// TIA Portal project "lab6" (V15)

(* hardware
DEVICE "S7-1200 station_1"  S7-1200 Station
   slot 0: "Rack_0"  S7-1200 Rack  Rack  V1.0
   slot 1: "PLC_1"  CPU 1214C DC/DC/DC  6ES7 214-1AG40-0XB0  V4.2
      slot 3: "AQ 1x12BIT_1"  AQ1 signal board  6ES7 232-4HA30-0XB0  V1.0
   slot 101: "CM 1243-5"  CM 1243-5  6GK7 243-5DX30-0XE0  V1.3
   slot 102: "CM 1241 (RS485)_1"  CM 1241 (RS485)  6ES7 241-1CH30-0XB0  V1.0
*)

// ===== PLC "PLC_1"  CPU 1214C DC/DC/DC =====

VAR_GLOBAL   // PLC tag table "Default tag table"
   "Tag_1" AT %I0.0 : Bool;
   "Tag_2" AT %MW10 : Int;
   "Tag_3" AT %Q0.5 : Bool;
   "Tag_4" AT %I0.1 : Bool;
   "Tag_5" AT %Q0.1 : Bool;
   "Tag_6" AT %Q0.2 : Bool;
   "System_Byte" AT %MB1 : Byte;
   "FirstScan" AT %M1.0 : Bool;
   "DiagStatusUpdate" AT %M1.1 : Bool;
   "AlwaysTRUE" AT %M1.2 : Bool;
   "AlwaysFALSE" AT %M1.3 : Bool;
   "Clock_Byte" AT %MB0 : Byte;
   "Clock_10Hz" AT %M0.0 : Bool;
   "Clock_5Hz" AT %M0.1 : Bool;
   "Clock_2.5Hz" AT %M0.2 : Bool;
   "Clock_2Hz" AT %M0.3 : Bool;
   "Clock_1.25Hz" AT %M0.4 : Bool;
   "Clock_1Hz" AT %M0.5 : Bool;
   "Clock_0.625Hz" AT %M0.6 : Bool;
   "Clock_0.5Hz" AT %M0.7 : Bool;
   "ZWIEKSZ" AT %I0.3 : Bool;
   "SPRZEZENIE" AT %M20.0 : Bool;
   "ANALOG" AT %MW24 : Word;
   "ZMNIEJSZ" AT %I0.4 : Bool;
   "START" AT %I0.6 : Bool;
END_VAR

// folder: System blocks/Program resources

DATA_BLOCK "licznikOsob"   // DB1
{ S7_Optimized_Access := 'TRUE' }
AUTHOR : Simatic
FAMILY : IEC
NAME : CNTR
VERSION : 1.0
// stored: InstanceOfName IEC_COUNTER
"IEC_COUNTER"
BEGIN
END_DATA_BLOCK

DATA_BLOCK "T1"   // DB2
{ S7_Optimized_Access := 'TRUE' }
AUTHOR : Simatic
FAMILY : IEC
NAME : IEC_TMR
VERSION : 1.0
// stored: InstanceOfName IEC_TIMER
"IEC_TIMER"
BEGIN
END_DATA_BLOCK

DATA_BLOCK "t2"   // DB3
{ S7_Optimized_Access := 'TRUE' }
AUTHOR : Simatic
FAMILY : IEC
NAME : IEC_TMR
VERSION : 1.0
// stored: InstanceOfName IEC_TIMER
"IEC_TIMER"
BEGIN
END_DATA_BLOCK

// folder: (top level)

ORGANIZATION_BLOCK "Main"   // OB1, LAD, ProgramCycle
TITLE = "Main Program Sweep (Cycle)"
{ S7_Optimized_Access := 'TRUE' }
VERSION : 0.1
   VAR_INPUT
      Initial_Call : Bool;   // Initial call of this OB
      Remanence : Bool;   // =True, if remanent data are available
   END_VAR
BEGIN

REGION Network 1: lICZNIK OSOB W POMIESZCZENIU
   // ZLICZA 7 OSOB
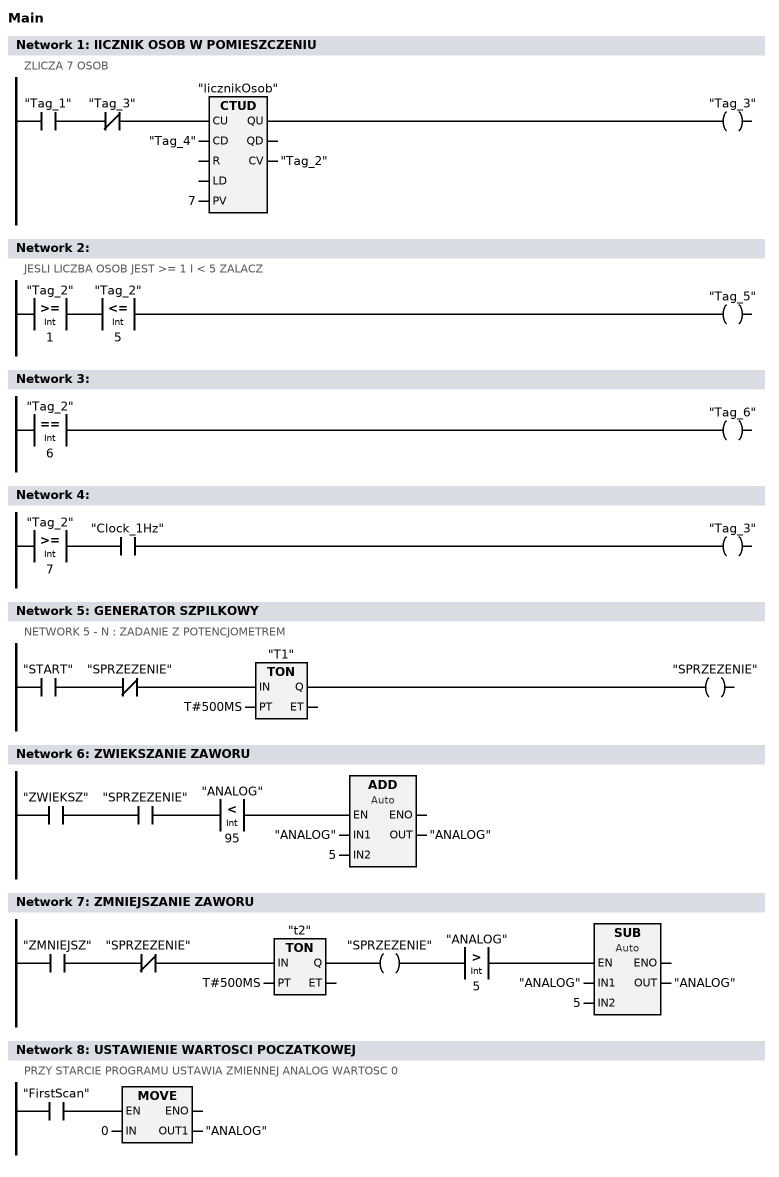
   "licznikOsob".CTUD(CU := "Tag_1" AND NOT "Tag_3", CD := "Tag_4", PV := 7, CV => "Tag_2");
   "Tag_3" := "licznikOsob".QU;
END_REGION

REGION Network 2
   // JESLI LICZBA OSOB JEST >= 1 I < 5 ZALACZ
   RUNG wire#powerrail
      { S7_Templates := "SrcType := Int" } GE_Contact(in1 := "Tag_2", in2 := 1)
      { S7_Templates := "SrcType := Int" } LE_Contact(in1 := "Tag_2", in2 := 5)
      Coil( "Tag_5" )
   END_RUNG
   // the same network as SCL:
   "Tag_5" := ("Tag_2" >= 1) AND ("Tag_2" <= 5);
END_REGION

REGION Network 3
   RUNG wire#powerrail
      { S7_Templates := "SrcType := Int" } EQ_Contact(in1 := "Tag_2", in2 := 6)
      Coil( "Tag_6" )
   END_RUNG
   // the same network as SCL:
   "Tag_6" := "Tag_2" = 6;
END_REGION

REGION Network 4
   RUNG wire#powerrail
      { S7_Templates := "SrcType := Int" } GE_Contact(in1 := "Tag_2", in2 := 7)
      Contact( "Clock_1Hz" )
      Coil( "Tag_3" )
   END_RUNG
   // the same network as SCL:
   "Tag_3" := ("Tag_2" >= 7) AND "Clock_1Hz";
END_REGION

REGION Network 5: GENERATOR SZPILKOWY
   // NETWORK 5 - N : ZADANIE Z POTENCJOMETREM
   "T1".TON(IN := "START" AND NOT "SPRZEZENIE", PT := T#500MS);
   "SPRZEZENIE" := "T1".Q;
END_REGION

REGION Network 6: ZWIEKSZANIE ZAWORU
   RUNG wire#powerrail
      Contact( "ZWIEKSZ" )
      Contact( "SPRZEZENIE" )
      { S7_Templates := "SrcType := Int" } LT_Contact(in1 := "ANALOG", in2 := 95)
      Add(in1 := "ANALOG", in2 := 5, out => "ANALOG")
   END_RUNG
   // the same network as SCL:
   IF "ZWIEKSZ" AND "SPRZEZENIE" AND ("ANALOG" < 95) THEN "ANALOG" := "ANALOG" + 5; END_IF;
END_REGION

REGION Network 7: ZMNIEJSZANIE ZAWORU
   "t2".TON(IN := "ZMNIEJSZ" AND NOT "SPRZEZENIE", PT := T#500MS);
   "SPRZEZENIE" := "t2".Q;
   IF "t2".Q AND ("ANALOG" > 5) THEN "ANALOG" := "ANALOG" - 5; END_IF;
END_REGION

REGION Network 8: USTAWIENIE WARTOSCI POCZATKOWEJ
   // PRZY STARCIE PROGRAMU USTAWIA ZMIENNEJ ANALOG WARTOSC 0
   RUNG wire#powerrail
      Contact( "FirstScan" )
      Move(in := 0, out1 => "ANALOG")
   END_RUNG
   // the same network as SCL:
   IF "FirstScan" THEN "ANALOG" := 0; END_IF;
END_REGION
END_ORGANIZATION_BLOCK